FUNCTION ConvertTimeToString : STRING
VAR_INPUT
	DataInput	: TIME;
END_VAR
VAR
END_VAR

ConvertTimeToString:=DELETE(TOD_TO_STRING(TIME_TO_TOD(DataInput)),5,0);

END_FUNCTION

(* stored: Version 1.1.0.1, ProductVersion 3.1.4024.12
   POU ConvertTimeToString: Id {ca112b8e-0b4a-423d-b40e-c9c8300e4ecf}, SpecialFunc None *)
